// Block: A0303_Spalla_Pers

DATA_BLOCK A0303_Spalla_Pers
VERSION : 0.1
   NON_RETAIN
   VAR
      Par : Struct
         Testa : Struct
            Ax : Positioning_DOL_Machine_Par;
            Ax_Pers : Positioning_DOL_Machine_Pers_Data;
            Enc : PosFbk_RTN;
         END_STRUCT;
         Coda : Struct
            Ax : Positioning_DOL_Machine_Par;
            Ax_Pers : Positioning_DOL_Machine_Pers_Data;
            Enc : PosFbk_RTN;
         END_STRUCT;
      END_STRUCT;
      Par_Mach_Testa : Struct
         MinDistanzaConParegg : LReal;
         ToleranceWindow : LReal;
      END_STRUCT;
      Par_Mach_Coda : Struct
         MinDistanzaConParegg : LReal;
         ToleranceWindow : LReal;
      END_STRUCT;
   END_VAR

BEGIN
   // No initialization required
END_DATA_BLOCK
